(* IEC 61131-3 sources: plc_simulator/services/codesys/POUs/SIM, 13 files *)

(* ---- SIM_FindStation.st ---- *)
(* ============================================================
 *  SIM_FindStation — Find a station by its number

   Company : Galvatek part of the John Cockerill Group
   Author  : Jarmo Piipponen
   Created : 25.03.2026
   ============================================================
   Direct lookup in Stations[] by station number.
   Returns x_mm (DINT); other fields via VAR_OUTPUT.
   ------------------------------------------------------------
   Changes:
   ============================================================ *)

FUNCTION SIM_FindStation : DINT   (* returns x_mm *)
VAR_INPUT
  station_number : INT;
END_VAR
VAR_OUTPUT
  found           : BOOL;
  skind           : INT;
  device_delay_s  : REAL;
  dropping_time_s : REAL;
END_VAR
VAR_EXTERNAL CONSTANT
    MIN_StationIndex : INT;
    MAX_StationIndex : INT;
END_VAR
VAR_EXTERNAL
  Stations : ARRAY[MIN_StationIndex..MAX_StationIndex] OF UDT_StationType;
END_VAR
VAR
  stn_data : UDT_StationType;
END_VAR

  (* Direct lookup by station number — no loop needed *)
  IF (station_number >= MIN_StationIndex) AND (station_number <= MAX_StationIndex) THEN
    stn_data := Stations[station_number];
    IF stn_data.TankId <> 0 THEN
      found := TRUE;
      SIM_FindStation := stn_data.XPosition;
      skind := stn_data.DryWet;
      device_delay_s := INT_TO_REAL(stn_data.DeviceDelay) / 10.0;
      dropping_time_s := INT_TO_REAL(stn_data.DrippingTime) / 10.0;
      RETURN;
    END_IF;
  END_IF;

  found := FALSE;
  SIM_FindStation := 0;
  skind := 0;
  device_delay_s := 0.0;
  dropping_time_s := 0.0;

END_FUNCTION

(* ---- FB_SIM_ClearConfig.st ---- *)
(* ============================================================
   FB_SIM_ClearConfig — Clear all PLC configuration data

   Company : Galvatek part of the John Cockerill Group
   Author  : Jarmo Piipponen
   Created : 25.03.2026
   ============================================================
   Called by PLC_PRG when Gateway sends cmd=3 (clear_all).
   Zeroes out all stations, transporter configs, transporter
   states and units so the PLC is ready for fresh config upload.
   ------------------------------------------------------------
   Changes:
   ============================================================ *)

FUNCTION_BLOCK FB_SIM_ClearConfig
VAR_EXTERNAL CONSTANT
    MAX_TRANSPORTERS    : INT;
    MAX_STATIONS_PER_STEP       : INT;
    MAX_STEPS_PER_PROGRAM       : INT;
    MAX_TASK_QUEUE      : INT;
    MIN_STATION_INDEX : INT;
    MAX_STATION_INDEX   : INT;
    MAX_UNITS           : INT;
    DEP_MAX_WAITING     : INT;
    NOT_PROCESSED       : INT;
END_VAR

VAR_EXTERNAL
  CountStations       : INT;
  Stations         : ARRAY[MIN_STATION_INDEX..MAX_STATION_INDEX] OF UDT_StationType;
  g_station_occupancy     : ARRAY[1..MAX_STATION_INDEX] OF UDT_JC_UnitAtStationType;
  Transporters              : ARRAY[0..MAX_TRANSPORTERS] OF UDT_TransporterType;
  g_transporter      : ARRAY[1..MAX_TRANSPORTERS] OF UDT_TransporterStatusType;
  g_sim_trans        : ARRAY[1..MAX_TRANSPORTERS] OF UDT_JC_SimTransporterType;
  g_dispatched_task  : ARRAY[1..MAX_TRANSPORTERS] OF UDT_JC_DispatchedTaskType;
  g_unit            : ARRAY[1..MAX_UNITS] OF UDT_JC_UnitType;
  g_ntt             : ARRAY[1..MAX_TRANSPORTERS] OF UDT_JC_NttTransporterType;
  g_batch          : ARRAY[1..MAX_UNITS] OF UDT_BatchType;
  TreatmentPrograms         : ARRAY[1..MAX_UNITS] OF UDT_TreatmentProgramType;
  g_avoid_status     : ARRAY[MIN_STATION_INDEX..MAX_STATION_INDEX] OF INT;
  g_schedule         : ARRAY[1..MAX_UNITS] OF UDT_JC_TskScheduleType;
  g_task             : ARRAY[1..MAX_TRANSPORTERS] OF UDT_JC_TskQueueType;
  g_sim_ui_schedule  : ARRAY[1..MAX_UNITS] OF UDT_JC_TskScheduleType;
  g_sim_ui_task      : ARRAY[1..MAX_TRANSPORTERS] OF UDT_JC_TskQueueType;
  g_sim_ui_wait_unit : INT;
  g_sim_ui_wait_reason : INT;
  g_dep_pending      : UDT_JC_DepPendingWriteType;
  g_dep_activated    : BOOL;
  g_tsk_stable       : BOOL;
  g_dep_waiting_count : INT;
  g_dep_waiting       : ARRAY[1..DEP_MAX_WAITING] OF INT;
END_VAR
VAR
  i : INT;
  j : INT;
  k : INT;
END_VAR

(* --- Clear all stations --- *)
FOR i := MIN_STATION_INDEX TO MAX_STATION_INDEX DO
  Stations[i].TankId       := 0;
  Stations[i].IsInUse       := FALSE;
  Stations[i].XPosition    := 0;
  Stations[i].YPosition    := 0;
  Stations[i].ZPosition    := 0;
  Stations[i].DryWet          := 0;
  Stations[i].StationType     := 0;
  Stations[i].DrippingTime := 0;
  Stations[i].DeviceDelay  := 0;
END_FOR;

(* --- Clear all vLocation tracking (transporters 1..MAX_TRANSPORTERS + stations MIN..MAX) --- *)
FOR i := 1 TO MAX_STATION_INDEX DO
  g_station_occupancy[i].UnitId     := 0;
  g_station_occupancy[i].ChangeTime := 0;
END_FOR;
CountStations := 0;

(* --- Clear all transporter configs --- *)
FOR i := 1 TO MAX_TRANSPORTERS DO
  Transporters[i].DrivePosMin   := 0;
  Transporters[i].DrivePosMax   := 0;
  Transporters[i].YMinDriveLimit   := 0;
  Transporters[i].YMaxDriveLimit   := 0;
  Transporters[i].CollisionWidth    := 0;
  Transporters[i].AvoidanceWidth    := 0;
  Transporters[i].Acceleration_X     := 0;
  Transporters[i].Deceleration_X     := 0;
  Transporters[i].SpeedMax_X    := 0;
  Transporters[i].ZPosDown    := 0;
  Transporters[i].ZPosSlowUp := 0;
  Transporters[i].ZPosSlowDown := 0;
  Transporters[i].ZPosSlowEnd := 0;
  Transporters[i].SpeedLiftSlow_Z   := 0;
  Transporters[i].SpeedLiftFast_Z   := 0;
  Transporters[i].DripTrayDelay  := 0;
  FOR j := 1 TO 4 DO
    Transporters[i].TaskArea[j].MinLift := 0;
    Transporters[i].TaskArea[j].MaxLift := 0;
    Transporters[i].TaskArea[j].MinSink := 0;
    Transporters[i].TaskArea[j].MaxSink := 0;
  END_FOR;
END_FOR;

(* --- Clear avoid status --- *)
FOR i := MIN_STATION_INDEX TO MAX_STATION_INDEX DO
  g_avoid_status[i] := 0;
END_FOR;

(* --- Clear all transporter states --- *)
FOR i := 1 TO MAX_TRANSPORTERS DO
  g_transporter[i].IsActive          := FALSE;
  g_transporter[i].Status          := 0;
  g_transporter[i].Phase           := 0;
  g_transporter[i].TaskId         := 0;
  g_transporter[i].LiftStationTarget    := 0;
  g_transporter[i].SinkStationTarget    := 0;
  g_transporter[i].DrippingTime   := 0;
  g_transporter[i].TaskRemainingTime  := 0;
  g_transporter[i].CurrentStation := 0;
  g_transporter[i].XFinalTarget  := 0;
  g_transporter[i].XDriveTarget  := 0;
  g_transporter[i].YFinalTarget  := 0;
  g_transporter[i].YDriveTarget  := 0;
  g_transporter[i].XPosition            := 0;
  g_transporter[i].YPosition            := 0;
  g_transporter[i].ZPosition            := 0;
  g_sim_trans[i].XVelocity           := 0;
  g_sim_trans[i].ZStage         := 0;
  g_sim_trans[i].ZTimer       := 0.0;
  g_transporter[i].IdleStartTime := g_time_s;  (* prevent spurious move-away after clear *)
  g_dispatched_task[i].Active := FALSE;
  g_transporter[i].XMinDriveLimit     := 0;
  g_transporter[i].XMaxDriveLimit     := 0;
END_FOR;

(* --- Clear all units --- *)
FOR i := 1 TO MAX_UNITS DO
  g_unit[i].vLocation := 0;
  g_unit[i].Status   := 0;
  g_unit[i].Target   := 0;
END_FOR;

(* --- Clear NTT destinations --- *)
FOR i := 1 TO MAX_TRANSPORTERS DO
  FOR j := 1 TO 8 DO
    g_ntt[i].Target[j].StationCount := 0;
    g_ntt[i].Target[j].FallbackCount := 0;
    FOR k := 1 TO MAX_STATIONS_PER_STEP DO
      g_ntt[i].Target[j].Stations[k] := 0;
      g_ntt[i].Target[j].FallbackStations[k] := 0;
    END_FOR;
  END_FOR;
END_FOR;

(* --- Clear all batches --- *)
FOR i := 1 TO MAX_UNITS DO
  g_batch[i].BatchCode  := 0;
  g_batch[i].State       := 0;
  g_batch[i].ProgId     := 0;
  g_batch[i].CurStage   := 0;
  g_batch[i].MinTime    := 0;
  g_batch[i].MaxTime    := 0;
  g_batch[i].CalTime    := 0;
  g_batch[i].StartTime  := LINT#0;
END_FOR;

(* --- Clear all treatment programs --- *)
FOR i := 1 TO MAX_UNITS DO
  TreatmentPrograms[i].ProgramId := 0;
  TreatmentPrograms[i].ProgramName := '';
  TreatmentPrograms[i].StepCount := 0;
  FOR j := 0 TO MAX_STEPS_PER_PROGRAM DO
    FOR k := 0 TO 4 DO
      TreatmentPrograms[i].Steps[j].Stations[k] := 0;
    END_FOR;
    TreatmentPrograms[i].Steps[j].StationCount := 0;
    TreatmentPrograms[i].Steps[j].MinTime := 0;
    TreatmentPrograms[i].Steps[j].MaxTime := 0;
    TreatmentPrograms[i].Steps[j].CalTime := 0;
  END_FOR;
END_FOR;

(* --- Clear all schedules (g_schedule) --- *)
FOR i := 1 TO MAX_UNITS DO
  g_schedule[i].StageCount := 0;
  FOR j := 0 TO MAX_STEPS_PER_PROGRAM DO
    g_schedule[i].Stages[j].Station       := 0;
    g_schedule[i].Stages[j].EntryTime    := 0;
    g_schedule[i].Stages[j].ExitTime     := 0;
    g_schedule[i].Stages[j].MinTime      := 0;
    g_schedule[i].Stages[j].CalcTime     := 0;
    g_schedule[i].Stages[j].MaxTime      := 0;
    g_schedule[i].Stages[j].TransferTime := 0;
  END_FOR;
END_FOR;

(* --- Clear all task queues (g_task) --- *)
FOR i := 1 TO MAX_TRANSPORTERS DO
  g_task[i].Count := 0;
  FOR j := 1 TO MAX_TASK_QUEUE DO
    g_task[i].Queue[j].Unit         := 0;
    g_task[i].Queue[j].Stage        := 0;
    g_task[i].Queue[j].LiftStationTarget := 0;
    g_task[i].Queue[j].SinkStationTarget := 0;
    g_task[i].Queue[j].StartTime   := 0;
    g_task[i].Queue[j].FinishTime  := 0;
    g_task[i].Queue[j].CalcTime    := 0;
    g_task[i].Queue[j].MinTime     := 0;
    g_task[i].Queue[j].MaxTime     := 0;
  END_FOR;
END_FOR;

(* --- Clear UI snapshot --- *)
FOR i := 1 TO MAX_UNITS DO
  g_sim_ui_schedule[i].StageCount := 0;
END_FOR;
FOR i := 1 TO MAX_TRANSPORTERS DO
  g_sim_ui_task[i].Count := 0;
END_FOR;
g_sim_ui_wait_unit := 0;
g_sim_ui_wait_reason := 0;

(* --- Clear departure pending write --- *)
g_dep_pending.Valid := FALSE;
g_dep_pending.BatchUnit  := 0;
g_dep_pending.BatchStage := 0;
g_dep_pending.BatchState := NOT_PROCESSED;

(* --- Clear departure scheduler state (previously missing) --- *)
g_dep_activated     := FALSE;
g_tsk_stable        := TRUE;   (* JS: tasksStableFlag starts true on empty line *)
g_dep_waiting_count := 0;
FOR i := 1 TO 5 DO
  g_dep_waiting[i] := 0;
END_FOR;

END_FUNCTION_BLOCK

(* ---- FB_SIM_EventQueue.st ---- *)
(* ============================================================
   FB_SIM_EventQueue — Event message queue handler (OPC UA)

   Company : Galvatek part of the John Cockerill Group
   Author  : Jarmo Piipponen
   Created : 25.03.2026
   ============================================================
   Manages a circular 10-slot event queue (g_event).

   Enqueue: caller writes msg to g_event_pending, sets
   g_event_pending_valid := TRUE. This FB picks it up.

   Dequeue: Gateway reads g_event.Buffer[Head] via OPC UA,
   then writes g_event_ack_seq to acknowledge.

   Called every PLC scan from PLC_PRG.
   ------------------------------------------------------------
   Changes:
   ============================================================ *)

FUNCTION_BLOCK FB_SIM_EventQueue
VAR_EXTERNAL
  g_event               : UDT_JC_EventQueueType;
  g_event_pending       : UDT_JC_EventMsgType;
  g_event_pending_valid : BOOL;
  g_event_ack_seq       : INT;
END_VAR
VAR
  vTail : INT;
END_VAR

(* ── 1. Enqueue: pick up pending message if queue not full ── *)
IF g_event_pending_valid AND g_event.Count < 10 THEN
  vTail := ((g_event.Head - 1 + g_event.Count) MOD 10) + 1;

  g_event_pending.Seq := g_event.NextSeq;
  g_event.NextSeq := g_event.NextSeq + 1;
  IF g_event.NextSeq > 32000 THEN
    g_event.NextSeq := 1;
  END_IF;

  g_event.Buffer[vTail] := g_event_pending;
  g_event.Count := g_event.Count + 1;

  g_event_pending_valid := FALSE;
END_IF;

(* ── 2. Dequeue: check gateway ack for head message ── *)
IF g_event.Count > 0 THEN
  IF g_event_ack_seq = g_event.Buffer[g_event.Head].Seq THEN
    g_event.Head := (g_event.Head MOD 10) + 1;
    g_event.Count := g_event.Count - 1;
  END_IF;
END_IF;

END_FUNCTION_BLOCK

(* ---- FB_SIM_MainCycle.st ---- *)
(* ===========================================================================================
 *  FB_SIM_MainCycle — Simulator main cycle (all SIM-specific logic)
 *
 *  Company : Galvatek part of the John Cockerill Group
 *  Author  : Jarmo Piipponen
 *  Created : 08.04.2026
 *
 * -------------------------------------------------------------------------------------------
 *  Encapsulates everything that is simulation-only and NOT vNeeded in production:
 *    - OPC UA command handler (init / clear)
 *    - System time calculation (g_time_s via offset from gateway sync)
 *    - TWA calculation
 *    - Physics simulation (delta_t + FB_SIM_RunTasks)
 *    - UI schedule snapshot for gateway
 *    - Event queue processing
 *
 *  In production PLC_PRG, this FB is removed entirely.
 *  PLC_PRG only needs: time from real PLC clock, TWA, MainScheduler.
 * ========================================================================================= *)

FUNCTION_BLOCK FB_SIM_MainCycle

(* Introduction of Variables ----------------------------------------------------------------*)

VAR_EXTERNAL CONSTANT
    MAX_TRANSPORTERS        : INT;
    MAX_STATIONS_PER_STEP   : INT;
    MIN_STATION_INDEX        : INT;
    MAX_STATION_INDEX        : INT;
    MAX_UNITS               : INT;
    DEP_MAX_WAITING         : INT;
END_VAR

VAR_EXTERNAL
  CountStations             : INT;
  Stations                  : ARRAY[MIN_STATION_INDEX..MAX_STATION_INDEX] OF UDT_StationType;
  g_station_occupancy       : ARRAY[1..MAX_STATION_INDEX] OF UDT_JC_UnitAtStationType;
  Transporters              : ARRAY[0..MAX_TRANSPORTERS] OF UDT_TransporterType;
  g_transporter             : ARRAY[1..MAX_TRANSPORTERS] OF UDT_TransporterStatusType;
  g_sim_trans               : ARRAY[1..MAX_TRANSPORTERS] OF UDT_JC_SimTransporterType;
  g_unit                    : ARRAY[1..MAX_UNITS] OF UDT_JC_UnitType;
  g_ntt                     : ARRAY[1..MAX_TRANSPORTERS] OF UDT_JC_NttTransporterType;
  g_batch                   : ARRAY[1..MAX_UNITS] OF UDT_BatchType;
  TreatmentPrograms         : ARRAY[1..MAX_UNITS] OF UDT_TreatmentProgramType;
  g_avoid_status            : ARRAY[MIN_STATION_INDEX..MAX_STATION_INDEX] OF INT;
  g_move                    : ARRAY[1..MAX_TRANSPORTERS] OF UDT_JC_MoveTimesType;
  g_schedule                : ARRAY[1..MAX_UNITS] OF UDT_JC_TskScheduleType;
  g_task                    : ARRAY[1..MAX_TRANSPORTERS] OF UDT_JC_TskQueueType;
  g_dep_activated           : BOOL;
  g_tsk_stable              : BOOL;
  g_dep_waiting_count       : INT;
  g_dep_overlap             : UDT_JC_DepOverlapType;
  g_dep_pending             : UDT_JC_DepPendingWriteType;
  g_dep_waiting             : ARRAY[1..DEP_MAX_WAITING] OF INT;
  g_sched_dbg_tsk_phase     : INT;
  g_sched_dbg_dep_phase     : INT;
  g_sim_ui_schedule         : ARRAY[1..MAX_UNITS] OF UDT_JC_TskScheduleType;
  g_sim_ui_task             : ARRAY[1..MAX_TRANSPORTERS] OF UDT_JC_TskQueueType;
  g_sim_ui_wait_unit        : INT;
  g_sim_ui_wait_reason      : INT;
  g_sched_dbg_turn          : INT;
  g_conflict_resolved       : BOOL;
  g_sched_dbg_batch_cnt     : INT;
  g_time_s                  : LINT;
  g_time_100ms              : LINT;
  g_time_offset             : LINT;
  g_time_sync               : LINT;
  g_event                   : UDT_JC_EventQueueType;
  g_event_pending           : UDT_JC_EventMsgType;
  g_event_pending_valid     : BOOL;
  g_event_ack_seq           : INT;
  g_cmd_code                : INT;
  g_cmd_param               : INT;
  g_sched_dbg_dep_cur_wait_unit : INT;
END_VAR

VAR_OUTPUT
  oInitDone               : BOOL;
END_VAR

VAR
  vInitDone                 : BOOL := FALSE;
  i                         : INT;
  vFB_ClearConfig                 : FB_SIM_ClearConfig;
  vFB_RunTasks                 : FB_SIM_RunTasks;
  vFB_EventQueue                 : FB_SIM_EventQueue;
  vNowMs                    : LINT := 0;
  vPrevMs                   : UDINT := 0;
  sim_delta_t               : REAL := 0.02;
  vPrevTskPhase            : INT := 0;
  vPrevDepPhase            : INT := 0;
END_VAR

(* ============================================================
   COMMAND HANDLER — OPC UA (direct, no sequence handshake)
   Gateway writes g_cmd_code + g_cmd_param in one atomic OPC UA
   call. PLC processes when g_cmd_code <> 0 and clears it.
   ============================================================ *)
IF g_cmd_code <> 0 THEN

  IF g_cmd_code = 3 THEN
    (* ── Clear all config data ── *)
    vFB_ClearConfig();
    vInitDone := FALSE;
    CountStations := 0;

  ELSIF g_cmd_code = 2 THEN
    (* ── Finish init: all config vAlready uploaded via OPC UA ── *)
    CountStations := g_cmd_param;

    FOR i := 1 TO MAX_TRANSPORTERS DO
      IF Transporters[i].TaskArea[1].MinLift > 0 THEN
        g_transporter[i].IsActive := TRUE;
        g_transporter[i].Status := 3;  (* auto_idle *)
      ELSE
        g_transporter[i].IsActive := FALSE;
        g_transporter[i].Status := 0;  (* not_used *)
      END_IF;
      g_transporter[i].Phase := 0;
      g_sim_trans[i].ZStage := 0;
      g_sim_trans[i].XVelocity := 0;
      g_sim_trans[i].ZTimer := 0.0;
      g_transporter[i].IdleStartTime := g_time_s;
      g_transporter[i].XMinDriveLimit := Transporters[i].DrivePosMin;
      g_transporter[i].XMaxDriveLimit := Transporters[i].DrivePosMax;

      (* Start position: at own vArea minimum, z=0 *)
      g_transporter[i].XPosition := Transporters[i].DrivePosMin;
      g_transporter[i].ZPosition := 0;
      g_transporter[i].CurrentStation := 0;
    END_FOR;

    vInitDone := TRUE;

    (* Calculate time offset: real unix time - uptime *)
    g_time_offset := g_time_sync - UDINT_TO_LINT(SysTimeGetMs()) / 1000;

    (* Build g_station_occupancy from g_unit[].vLocation so FB_SIM_RunTasks
       can find units on stations via g_station_occupancy[stn].UnitId.
       Gateway writes g_unit[] but not g_station_occupancy[]. *)
    FOR i := 1 TO MAX_UNITS DO
      IF g_unit[i].vLocation >= MIN_STATION_INDEX
         AND g_unit[i].vLocation <= MAX_STATION_INDEX THEN
        g_station_occupancy[g_unit[i].vLocation].UnitId     := i;
        g_station_occupancy[g_unit[i].vLocation].ChangeTime  := g_time_s;
      END_IF;
    END_FOR;

    (* Init event queue *)
    g_event.Head := 1;
    g_event.NextSeq := 1;
    g_event.Count := 0;
  END_IF;

  g_cmd_code := 0;  (* Command processed — clear trigger *)
END_IF;

(* ============================================================
   MAIN TRANSPORT CYCLE — only runs when vInitDone
   ============================================================ *)
IF vInitDone THEN

  (* ── System time: uptime + offset = real unix seconds ── *)
  vNowMs := UDINT_TO_LINT(SysTimeGetMs());
  g_time_s := g_time_offset + vNowMs / 1000;        (* seconds, unix epoch *)
  g_time_100ms := g_time_offset * 10 + vNowMs / 100; (* 0.1s ticks, unix epoch *)

  (* ── Actual cycle time for physics simulation ── *)
  IF vPrevMs > 0 THEN
    sim_delta_t := UDINT_TO_REAL(LINT_TO_UDINT(vNowMs) - vPrevMs) / 1000.0;
  END_IF;
  vPrevMs := LINT_TO_UDINT(vNowMs);

  (* ── Execute transporter tasks (physics simulation) ── *)
  vFB_RunTasks(iRun := vInitDone, iDeltaT := sim_delta_t);

END_IF;  (* vInitDone *)

oInitDone := vInitDone;

(* ── UI schedule snapshot — copy stable data for gateway reads ── *)
IF g_sched_dbg_tsk_phase = 10000 AND vPrevTskPhase <> 10000 THEN
  g_sim_ui_schedule := g_schedule;
  g_sim_ui_task     := g_task;
END_IF;
IF g_sched_dbg_dep_phase = 8000 AND vPrevDepPhase <> 8000 THEN
  g_sim_ui_wait_unit   := 0;
  g_sim_ui_wait_reason := 0;
END_IF;
IF g_sched_dbg_dep_phase = 9000 AND vPrevDepPhase <> 9000 THEN
  g_sim_ui_wait_unit   := g_sched_dbg_dep_cur_wait_unit;
  g_sim_ui_wait_reason := 1;
END_IF;
vPrevTskPhase := g_sched_dbg_tsk_phase;
vPrevDepPhase := g_sched_dbg_dep_phase;

(* ── Event queue — always runs, not gated by vInitDone ── *)
vFB_EventQueue();

END_FUNCTION_BLOCK

(* ---- FB_SIM_RunTasks.st ---- *)
(* ============================================================
   FB_SIM_RunTasks — Simulate transporter task execution

   Company : Galvatek part of the John Cockerill Group
   Author  : Jarmo Piipponen
   Created : 25.03.2026
   ============================================================
   For each active transporter [1..3], checks whether a new task
   has been assigned (task_id <> running_task_id) and executes
   the full transport cycle:

     Phase 0  idle        — waiting for new task
     Phase 1  to_lift     — X-drive towards lift station
     Phase 2  lifting     — Z-lift sequence (stages 1-5)
     Phase 3  to_sink     — X-drive towards sink station
     Phase 4  sinking     — Z-sink sequence (stages 6-8)

   Also maintains current_station (nearest station) every cycle.
   Called once per PLC scan from PLC_PRG.
   ------------------------------------------------------------
   Changes:
   ============================================================ *)

FUNCTION_BLOCK FB_SIM_RunTasks
VAR_INPUT
  iRun     : BOOL;   (* enable — typically vInitDone *)
  iDeltaT : REAL;   (* actual cycle time in seconds *)
END_VAR
VAR_EXTERNAL CONSTANT
    MAX_TRANSPORTERS    : INT;
    MAX_UNITS           : INT;
    MAX_STEPS_PER_PROGRAM          : INT;
    MIN_STATION_INDEX : INT;
    MAX_STATION_INDEX   : INT;
    IN_PROCESS          : INT;
END_VAR

VAR_EXTERNAL
  g_transporter  : ARRAY[1..MAX_TRANSPORTERS] OF UDT_TransporterStatusType;
  g_sim_trans    : ARRAY[1..MAX_TRANSPORTERS] OF UDT_JC_SimTransporterType;
  Stations      : ARRAY[MIN_STATION_INDEX..MAX_STATION_INDEX] OF UDT_StationType;
  g_station_occupancy  : ARRAY[1..MAX_STATION_INDEX] OF UDT_JC_UnitAtStationType;
  Transporters          : ARRAY[0..MAX_TRANSPORTERS] OF UDT_TransporterType;
  g_move         : ARRAY[1..MAX_TRANSPORTERS] OF UDT_JC_MoveTimesType;
  g_actual_move  : ARRAY[1..MAX_TRANSPORTERS] OF UDT_JC_ActualMoveTimeType;
  g_unit         : ARRAY[1..MAX_UNITS] OF UDT_JC_UnitType;
  g_batch        : ARRAY[1..MAX_UNITS] OF UDT_BatchType;
  TreatmentPrograms      : ARRAY[1..MAX_UNITS] OF UDT_TreatmentProgramType;
  g_time_s       : LINT;
  g_event_pending       : UDT_JC_EventMsgType;
  g_event_pending_valid : BOOL;
  g_dispatched_task     : ARRAY[1..MAX_TRANSPORTERS] OF UDT_JC_DispatchedTaskType;
END_VAR
VAR
  i            : INT;
  vIdx          : INT;
  (* Physics FB instances — one per transporter (MATIEC needs separate instances) *)
  fb_x1        : FB_SIM_XMotion;
  fb_x2        : FB_SIM_XMotion;
  fb_x3        : FB_SIM_XMotion;
  fb_z1        : FB_SIM_ZMotion;
  fb_z2        : FB_SIM_ZMotion;
  fb_z3        : FB_SIM_ZMotion;
  (* Temp vars for VAR_IN_OUT passing *)
  vTmpX        : DINT;
  vTmpVx       : DINT;
  vTmpZ        : DINT;
  vTmpZs       : INT;
  vTmpZt       : REAL;
  arrived_x    : BOOL;
  at_station   : BOOL;    (* TRUE only when actually at station, not just at drive limit *)
  arrived_z    : BOOL;
  vStationKind : INT;
  device_delay : REAL;
  vDropTime    : REAL;
  vPickUnitId : INT;     (* unit_id picked up from lift station *)
  vXferTotal   : REAL;    (* transfer time for UI progress bar *)
  vSinkUnitId : INT;     (* unit_id being placed at sink station *)
  (* Nearest-station calculation *)
  vNearestNum  : INT;
  vMinDist     : DINT;
  dx           : DINT;
  (* Actual move time tracker — now FC FC_STC_TrackMoveTimes, no instance vNeeded *)
  (* Unit vLocation update — now FC FC_STC_UpdateUnitLocation, no instance vNeeded *)
  (* Event helpers *)
  evt_unit     : INT;
  evt_diff     : LINT;
  (* Treatment time wait *)
  vCanLift       : BOOL;
  vLiftUid       : INT;      (* unit at lift station *)
  treat_cal      : DINT;      (* treatment cal_time for current stage *)
  treat_elapsed  : LINT;     (* seconds spent at lift station *)
  (* ── TASK_COMPLETE event: vPhase timestamps per transporter ── *)
  ts_task_start  : ARRAY[1..3] OF LINT;  (* Phase 0→1: task accepted *)
  ts_at_lift     : ARRAY[1..3] OF LINT;  (* Phase 1 at_station: arrived at lift *)
  ts_lift_begin  : ARRAY[1..3] OF LINT;  (* Phase 1→2: vCanLift, begin lift *)
  ts_lift_done   : ARRAY[1..3] OF LINT;  (* Phase 2→3: lift complete *)
  ts_at_sink     : ARRAY[1..3] OF LINT;  (* Phase 3→4: arrived at sink *)
  (* TASK_COMPLETE temp vars *)
  dd_lift_s      : INT;   (* lift device_delay in seconds *)
  dropping_s     : INT;   (* dropping/valutus time in seconds *)
  trip_s         : INT;   (* drip tray vDelay in seconds, 0 if not used *)
  vDurNosto      : INT;   (* computed nosto vDuration *)
  vDurLasku      : INT;   (* computed lasku vDuration *)
END_VAR

IF NOT iRun THEN
  RETURN;
END_IF;

FOR i := 1 TO MAX_TRANSPORTERS DO
  IF g_transporter[i].IsActive THEN

  (* ── Phase 0 → 1: Accept new task ───────────────────────── *)
  IF (g_transporter[i].Phase = 0)
     AND g_dispatched_task[i].Active THEN
    g_transporter[i].XFinalTarget := g_dispatched_task[i].LiftX;
    g_transporter[i].Status := 4;  (* auto_run — must be set before TrackMoveTimes *)
    g_transporter[i].Phase := 1;
    FC_STC_TrackMoveTimes(iTrans := i, iPrev := 0, iNew := 1);
    g_sim_trans[i].ZStage := 0;
    g_sim_trans[i].ZTimer := 0.0;
    (* Record task start timestamp *)
    ts_task_start[i] := g_time_s;
    ts_at_lift[i]    := LINT#0;

  (* ── Phase 1: Drive X towards lift station ──────────────── *)
  ELSIF g_transporter[i].Phase = 1 THEN
    vTmpX  := g_transporter[i].XPosition;
    vTmpVx := g_sim_trans[i].XVelocity;
    IF i = 1 THEN
      fb_x1(
        delta_t  := iDeltaT,
        x_target := g_transporter[i].XFinalTarget,
        x_min    := g_transporter[i].XMinDriveLimit,
        x_max    := g_transporter[i].XMaxDriveLimit,
        v_max    := Transporters[i].SpeedMax_X,
        t_acc    := Transporters[i].Acceleration_X,
        t_dec    := Transporters[i].Deceleration_X,
        x_pos    := vTmpX,
        v_x      := vTmpVx
      );
      arrived_x := fb_x1.arrived;
      g_transporter[i].XDriveTarget := fb_x1.x_drive;
    ELSIF i = 2 THEN
      fb_x2(
        delta_t  := iDeltaT,
        x_target := g_transporter[i].XFinalTarget,
        x_min    := g_transporter[i].XMinDriveLimit,
        x_max    := g_transporter[i].XMaxDriveLimit,
        v_max    := Transporters[i].SpeedMax_X,
        t_acc    := Transporters[i].Acceleration_X,
        t_dec    := Transporters[i].Deceleration_X,
        x_pos    := vTmpX,
        v_x      := vTmpVx
      );
      arrived_x := fb_x2.arrived;
      g_transporter[i].XDriveTarget := fb_x2.x_drive;
    ELSIF i = 3 THEN
      fb_x3(
        delta_t  := iDeltaT,
        x_target := g_transporter[i].XFinalTarget,
        x_min    := g_transporter[i].XMinDriveLimit,
        x_max    := g_transporter[i].XMaxDriveLimit,
        v_max    := Transporters[i].SpeedMax_X,
        t_acc    := Transporters[i].Acceleration_X,
        t_dec    := Transporters[i].Deceleration_X,
        x_pos    := vTmpX,
        v_x      := vTmpVx
      );
      arrived_x := fb_x3.arrived;
      g_transporter[i].XDriveTarget := fb_x3.x_drive;
    END_IF;
    g_transporter[i].XPosition  := vTmpX;
    g_sim_trans[i].XVelocity := vTmpVx;

    (* Only transition when actually at station, not just at drive limit *)
    at_station := arrived_x
                  AND (ABS(g_transporter[i].XPosition - g_transporter[i].XFinalTarget) <= 6);
    IF at_station THEN
      g_transporter[i].CurrentStation := g_transporter[i].LiftStationTarget;

      (* ── Move-away arrival: Status=3 means idle repositioning, not a real task ── *)
      IF g_transporter[i].Status = 3 THEN
        g_transporter[i].Phase := 0;
        g_transporter[i].IdleStartTime := g_time_s;
        FC_STC_TrackMoveTimes(iTrans := i, iPrev := 1, iNew := 0);
      ELSE
      (* Record arrival at lift station (first time only) *)
      IF ts_at_lift[i] = LINT#0 THEN
        ts_at_lift[i] := g_time_s;
      END_IF;

      (* ── Wait for treatment time AND device_delay before lifting ──
         Z-movement starts when the LONGER of two has elapsed:
         1. Remaining treatment time (unit must finish treatment)
         2. Station device_delay (vCovers must be open)
         Both timers run simultaneously from transporter arrival.
         This matches JS behavior: max(treatment, device_delay). *)
      vCanLift := TRUE;
      device_delay := INT_TO_REAL(g_dispatched_task[i].LiftDeviceDelay_x10) / 10.0;
      vDropTime := INT_TO_REAL(g_dispatched_task[i].DroppingTime_x10) / 10.0;

      (* Check treatment time *)
      vLiftUid := g_station_occupancy[g_transporter[i].LiftStationTarget].UnitId;
      IF vLiftUid >= 1 AND vLiftUid <= MAX_UNITS THEN
        IF g_batch[vLiftUid].State = IN_PROCESS
           AND g_batch[vLiftUid].CurStage >= 1
           AND g_batch[vLiftUid].CurStage <= MAX_STEPS_PER_PROGRAM THEN
          treat_cal := TreatmentPrograms[vLiftUid].Steps[g_batch[vLiftUid].CurStage].CalTime;
          IF treat_cal > 0 THEN
            treat_elapsed := g_time_s - g_station_occupancy[g_transporter[i].LiftStationTarget].ChangeTime;
            IF treat_elapsed < DINT_TO_LINT(treat_cal) THEN
              vCanLift := FALSE;
            END_IF;
          END_IF;
        END_IF;
      END_IF;

      (* Check device_delay — vCovers must have had time to open since arrival *)
      IF vCanLift AND device_delay > 0.0 THEN
        IF LINT_TO_REAL(g_time_s - ts_at_lift[i]) < device_delay THEN
          vCanLift := FALSE;
        END_IF;
      END_IF;

      IF vCanLift THEN
      (* Record lift begin timestamp *)
      ts_lift_begin[i] := g_time_s;
      (* vDropTime vAlready captured by STC_FindStation above *)
      (* Skip stage 1 — device_delay vAlready overlapped above.
         Z-movement starts immediately (stage 2).
         dropping_time and drip_tray_delay happen at the TOP. *)
      g_transporter[i].ZPosition := 0;
      g_sim_trans[i].ZTimer := 0.0;
      g_sim_trans[i].ZStage := 2;
      g_transporter[i].Phase := 2;
      FC_STC_TrackMoveTimes(iTrans := i, iPrev := 1, iNew := 2);

      (* ── Calculate transfer time (used by event + batch times) ── *)
      vXferTotal := DINT_TO_REAL(g_dispatched_task[i].TransferTime_x10) / 10.0;
      IF vXferTotal < 5.0 THEN vXferTotal := 60.0; END_IF;

      (* ── Emit LIFT event (msg_type=2) ── *)
      evt_unit := g_station_occupancy[g_transporter[i].LiftStationTarget].UnitId;
      IF NOT g_event_pending_valid AND evt_unit >= 1 THEN
        g_event_pending.MsgType := 2;
        g_event_pending.TsHi := LINT_TO_UINT(g_time_s / LINT#65536);
        g_event_pending.TsLo := LINT_TO_UINT(g_time_s MOD LINT#65536);
        g_event_pending.Payload[1]  := LINT_TO_INT(g_transporter[i].TaskId / LINT#65536);   (* TaskId_Hi *)
        g_event_pending.Payload[2]  := LINT_TO_INT(g_transporter[i].TaskId MOD LINT#65536);  (* TaskId_Lo *)
        g_event_pending.Payload[3]  := i;
        g_event_pending.Payload[4]  := evt_unit;
        g_event_pending.Payload[5]  := g_transporter[i].LiftStationTarget;
        g_event_pending.Payload[6]  := g_batch[evt_unit].BatchCode;
        g_event_pending.Payload[7]  := g_batch[evt_unit].CurStage;
        evt_diff := g_time_s - g_station_occupancy[g_transporter[i].LiftStationTarget].ChangeTime;
        IF evt_diff > LINT#32000 THEN
          g_event_pending.Payload[8] := 32000;
        ELSE
          g_event_pending.Payload[8] := LINT_TO_INT(evt_diff);
        END_IF;
        (* ── Original program calc/min/max for this stage ── *)
        (* g_sim_trans holds dispatch-time scheduler values which may differ
           from the treatment program originals. Read directly from TreatmentPrograms
           using the batch's current stage (CurStage=1-based program index). *)
        IF g_batch[evt_unit].CurStage >= 1 AND g_batch[evt_unit].CurStage <= 30 THEN
          g_event_pending.Payload[9]  := DINT_TO_INT(TreatmentPrograms[evt_unit].Steps[g_batch[evt_unit].CurStage].CalTime);
          g_event_pending.Payload[10] := DINT_TO_INT(TreatmentPrograms[evt_unit].Steps[g_batch[evt_unit].CurStage].MinTime);
          g_event_pending.Payload[11] := DINT_TO_INT(TreatmentPrograms[evt_unit].Steps[g_batch[evt_unit].CurStage].MaxTime);
        ELSE
          (* Stage 0 (pickup) — no program step *)
          g_event_pending.Payload[9]  := 0;
          g_event_pending.Payload[10] := 0;
          g_event_pending.Payload[11] := 0;
        END_IF;
        g_event_pending.Payload[12] := REAL_TO_INT(vXferTotal);
        g_event_pending_valid := TRUE;
      END_IF;

      (* Unit moves from lift station → transporter *)
      vPickUnitId := g_station_occupancy[g_transporter[i].LiftStationTarget].UnitId;
      IF vPickUnitId >= 1 THEN
        FC_STC_UpdateUnitLocation(iUnit := vPickUnitId, iLocation := i, iNttPrimary := 0);

        (* Set batch transfer times for UI progress bar — matches JS behavior *)
        g_batch[vPickUnitId].StartTime := g_time_s;
        g_batch[vPickUnitId].CalTime   := REAL_TO_DINT(vXferTotal);
        g_batch[vPickUnitId].MinTime   := g_batch[vPickUnitId].CalTime;
        g_batch[vPickUnitId].MaxTime   := 600;
      END_IF;
      END_IF;  (* vCanLift *)
      END_IF;  (* Status=3 ELSE branch *)
    END_IF;
    (* If arrived_x but not at_station → at drive limit, wait for clearance *)

  (* ── Phase 2: Lift Z at lift station ────────────────────── *)
  ELSIF g_transporter[i].Phase = 2 THEN
    vStationKind := g_dispatched_task[i].LiftKind;
    vTmpZ  := g_transporter[i].ZPosition;
    vTmpZs := g_sim_trans[i].ZStage;
    vTmpZt := g_sim_trans[i].ZTimer;
    IF i = 1 THEN
      fb_z1(
        delta_t       := iDeltaT,
        vStationKind  := vStationKind,
        ZPosDown        := Transporters[i].ZPosDown,
        ZPosUp          := 0,
        ZPosSlowUp      := Transporters[i].ZPosSlowUp,
        ZPosSlowDown    := Transporters[i].ZPosSlowDown,
        ZPosSlowEnd     := Transporters[i].ZPosSlowEnd,
        SpeedLiftSlow_Z := Transporters[i].SpeedLiftSlow_Z,
        SpeedLiftFast_Z := Transporters[i].SpeedLiftFast_Z,
        DripTrayDelay   := Transporters[i].DripTrayDelay,
        DroppingTime    := g_dispatched_task[i].DroppingTime_x10,
        z_mm          := vTmpZ,
        z_stage       := vTmpZs,
        z_timer_s     := vTmpZt
      );
      arrived_z := fb_z1.vDone;
    ELSIF i = 2 THEN
      fb_z2(
        delta_t       := iDeltaT,
        vStationKind  := vStationKind,
        ZPosDown        := Transporters[i].ZPosDown,
        ZPosUp          := 0,
        ZPosSlowUp      := Transporters[i].ZPosSlowUp,
        ZPosSlowDown    := Transporters[i].ZPosSlowDown,
        ZPosSlowEnd     := Transporters[i].ZPosSlowEnd,
        SpeedLiftSlow_Z := Transporters[i].SpeedLiftSlow_Z,
        SpeedLiftFast_Z := Transporters[i].SpeedLiftFast_Z,
        DripTrayDelay   := Transporters[i].DripTrayDelay,
        DroppingTime    := g_dispatched_task[i].DroppingTime_x10,
        z_mm          := vTmpZ,
        z_stage       := vTmpZs,
        z_timer_s     := vTmpZt
      );
      arrived_z := fb_z2.vDone;
    ELSIF i = 3 THEN
      fb_z3(
        delta_t       := iDeltaT,
        vStationKind  := vStationKind,
        ZPosDown        := Transporters[i].ZPosDown,
        ZPosUp          := 0,
        ZPosSlowUp      := Transporters[i].ZPosSlowUp,
        ZPosSlowDown    := Transporters[i].ZPosSlowDown,
        ZPosSlowEnd     := Transporters[i].ZPosSlowEnd,
        SpeedLiftSlow_Z := Transporters[i].SpeedLiftSlow_Z,
        SpeedLiftFast_Z := Transporters[i].SpeedLiftFast_Z,
        DripTrayDelay   := Transporters[i].DripTrayDelay,
        DroppingTime    := g_dispatched_task[i].DroppingTime_x10,
        z_mm          := vTmpZ,
        z_stage       := vTmpZs,
        z_timer_s     := vTmpZt
      );
      arrived_z := fb_z3.vDone;
    END_IF;
    g_transporter[i].ZPosition      := vTmpZ;
    g_sim_trans[i].ZStage   := vTmpZs;
    g_sim_trans[i].ZTimer := vTmpZt;
    IF arrived_z THEN
      (* Record lift vDone timestamp *)
      ts_lift_done[i] := g_time_s;
      g_transporter[i].XFinalTarget := g_dispatched_task[i].SinkX;
      g_transporter[i].Phase := 3;
      FC_STC_TrackMoveTimes(iTrans := i, iPrev := 2, iNew := 3);
    END_IF;

  (* ── Phase 3: Drive X towards sink station ─────────────── *)
  ELSIF g_transporter[i].Phase = 3 THEN
    vTmpX  := g_transporter[i].XPosition;
    vTmpVx := g_sim_trans[i].XVelocity;
    IF i = 1 THEN
      fb_x1(
        delta_t  := iDeltaT,
        x_target := g_transporter[i].XFinalTarget,
        x_min    := g_transporter[i].XMinDriveLimit,
        x_max    := g_transporter[i].XMaxDriveLimit,
        v_max    := Transporters[i].SpeedMax_X,
        t_acc    := Transporters[i].Acceleration_X,
        t_dec    := Transporters[i].Deceleration_X,
        x_pos    := vTmpX,
        v_x      := vTmpVx
      );
      arrived_x := fb_x1.arrived;
      g_transporter[i].XDriveTarget := fb_x1.x_drive;
    ELSIF i = 2 THEN
      fb_x2(
        delta_t  := iDeltaT,
        x_target := g_transporter[i].XFinalTarget,
        x_min    := g_transporter[i].XMinDriveLimit,
        x_max    := g_transporter[i].XMaxDriveLimit,
        v_max    := Transporters[i].SpeedMax_X,
        t_acc    := Transporters[i].Acceleration_X,
        t_dec    := Transporters[i].Deceleration_X,
        x_pos    := vTmpX,
        v_x      := vTmpVx
      );
      arrived_x := fb_x2.arrived;
      g_transporter[i].XDriveTarget := fb_x2.x_drive;
    ELSIF i = 3 THEN
      fb_x3(
        delta_t  := iDeltaT,
        x_target := g_transporter[i].XFinalTarget,
        x_min    := g_transporter[i].XMinDriveLimit,
        x_max    := g_transporter[i].XMaxDriveLimit,
        v_max    := Transporters[i].SpeedMax_X,
        t_acc    := Transporters[i].Acceleration_X,
        t_dec    := Transporters[i].Deceleration_X,
        x_pos    := vTmpX,
        v_x      := vTmpVx
      );
      arrived_x := fb_x3.arrived;
      g_transporter[i].XDriveTarget := fb_x3.x_drive;
    END_IF;
    g_transporter[i].XPosition  := vTmpX;
    g_sim_trans[i].XVelocity := vTmpVx;

    (* Only transition when actually at station, not just at drive limit *)
    at_station := arrived_x
                  AND (ABS(g_transporter[i].XPosition - g_transporter[i].XFinalTarget) <= 6);
    IF at_station THEN
      g_transporter[i].CurrentStation := g_transporter[i].SinkStationTarget;
      (* Record arrival at sink timestamp *)
      ts_at_sink[i] := g_time_s;
      device_delay := INT_TO_REAL(g_dispatched_task[i].SinkDeviceDelay_x10) / 10.0;
      g_sim_trans[i].ZTimer := device_delay + INT_TO_REAL(g_dispatched_task[i].DripTrayDelay_x10) / 10.0;
      g_sim_trans[i].ZStage := 6;
      g_transporter[i].Phase := 4;
      FC_STC_TrackMoveTimes(iTrans := i, iPrev := 3, iNew := 4);
    END_IF;
    (* If arrived_x but not at_station → at drive limit, wait for clearance *)

  (* ── Phase 4: Sink Z at sink station ───────────────────── *)
  ELSIF g_transporter[i].Phase = 4 THEN
    vStationKind := g_dispatched_task[i].SinkKind;
    vTmpZ  := g_transporter[i].ZPosition;
    vTmpZs := g_sim_trans[i].ZStage;
    vTmpZt := g_sim_trans[i].ZTimer;
    IF i = 1 THEN
      fb_z1(
        delta_t       := iDeltaT,
        vStationKind  := vStationKind,
        ZPosDown        := Transporters[i].ZPosDown,
        ZPosUp          := 0,
        ZPosSlowUp      := Transporters[i].ZPosSlowUp,
        ZPosSlowDown    := Transporters[i].ZPosSlowDown,
        ZPosSlowEnd     := Transporters[i].ZPosSlowEnd,
        SpeedLiftSlow_Z := Transporters[i].SpeedLiftSlow_Z,
        SpeedLiftFast_Z := Transporters[i].SpeedLiftFast_Z,
        DripTrayDelay   := Transporters[i].DripTrayDelay,
        DroppingTime    := 0,
        z_mm          := vTmpZ,
        z_stage       := vTmpZs,
        z_timer_s     := vTmpZt
      );
      arrived_z := fb_z1.vDone;
    ELSIF i = 2 THEN
      fb_z2(
        delta_t       := iDeltaT,
        vStationKind  := vStationKind,
        ZPosDown        := Transporters[i].ZPosDown,
        ZPosUp          := 0,
        ZPosSlowUp      := Transporters[i].ZPosSlowUp,
        ZPosSlowDown    := Transporters[i].ZPosSlowDown,
        ZPosSlowEnd     := Transporters[i].ZPosSlowEnd,
        SpeedLiftSlow_Z := Transporters[i].SpeedLiftSlow_Z,
        SpeedLiftFast_Z := Transporters[i].SpeedLiftFast_Z,
        DripTrayDelay   := Transporters[i].DripTrayDelay,
        DroppingTime    := 0,
        z_mm          := vTmpZ,
        z_stage       := vTmpZs,
        z_timer_s     := vTmpZt
      );
      arrived_z := fb_z2.vDone;
    ELSIF i = 3 THEN
      fb_z3(
        delta_t       := iDeltaT,
        vStationKind  := vStationKind,
        ZPosDown        := Transporters[i].ZPosDown,
        ZPosUp          := 0,
        ZPosSlowUp      := Transporters[i].ZPosSlowUp,
        ZPosSlowDown    := Transporters[i].ZPosSlowDown,
        ZPosSlowEnd     := Transporters[i].ZPosSlowEnd,
        SpeedLiftSlow_Z := Transporters[i].SpeedLiftSlow_Z,
        SpeedLiftFast_Z := Transporters[i].SpeedLiftFast_Z,
        DripTrayDelay   := Transporters[i].DripTrayDelay,
        DroppingTime    := 0,
        z_mm          := vTmpZ,
        z_stage       := vTmpZs,
        z_timer_s     := vTmpZt
      );
      arrived_z := fb_z3.vDone;
    END_IF;
    g_transporter[i].ZPosition      := vTmpZ;
    g_sim_trans[i].ZStage   := vTmpZs;
    g_sim_trans[i].ZTimer := vTmpZt;
    IF arrived_z THEN
      (* ── Emit TASK_COMPLETE event (msg_type=3) before Phase reset ── *)
      IF NOT g_event_pending_valid THEN
        (* Config-based sub-vPhase durations *)
        dropping_s := g_transporter[i].DrippingTime / 10;
        IF Transporters[i].DripTrayInUse THEN
          trip_s := Transporters[i].DripTrayDelay / 10;
        ELSE
          trip_s := 0;
        END_IF;
        (* Nosto = total lift vPhase - dropping - trip_close
           device_delay no longer in lift vPhase (overlapped in Phase 1) *)
        vDurNosto := LINT_TO_INT(ts_lift_done[i] - ts_lift_begin[i])
                     - dropping_s - trip_s;
        IF vDurNosto < 0 THEN vDurNosto := 0; END_IF;
        (* Lasku = total sink vPhase - device_delay - trip_open *)
        dd_lift_s := g_dispatched_task[i].SinkDeviceDelay_x10 / 10;
        vDurLasku := LINT_TO_INT(g_time_s - ts_at_sink[i]) - dd_lift_s - trip_s;
        IF vDurLasku < 0 THEN vDurLasku := 0; END_IF;

        g_event_pending.MsgType := 3;
        g_event_pending.TsHi := LINT_TO_UINT(g_time_s / LINT#65536);
        g_event_pending.TsLo := LINT_TO_UINT(g_time_s MOD LINT#65536);
        g_event_pending.Payload[1]  := LINT_TO_INT(g_transporter[i].TaskId / LINT#65536);   (* TaskId_Hi *)
        g_event_pending.Payload[2]  := LINT_TO_INT(g_transporter[i].TaskId MOD LINT#65536);  (* TaskId_Lo *)
        g_event_pending.Payload[3]  := i;                                                     (* transporter *)
        g_event_pending.Payload[4]  := LINT_TO_INT(ts_at_lift[i] - ts_task_start[i]);         (* siirto nostoasemalle *)
        g_event_pending.Payload[5]  := LINT_TO_INT(ts_lift_begin[i] - ts_at_lift[i]);         (* odotus ennen nostoa (max(treat,dev_delay)) *)
        g_event_pending.Payload[6]  := vDurNosto;                                             (* nosto *)
        g_event_pending.Payload[7]  := dropping_s;                                            (* valutus *)
        g_event_pending.Payload[8]  := trip_s;                                                (* trip close *)
        g_event_pending.Payload[9]  := LINT_TO_INT(ts_at_sink[i] - ts_lift_done[i]);          (* siirto laskuasemalle *)
        g_event_pending.Payload[10] := trip_s;                                                (* trip open *)
        g_event_pending.Payload[11] := vDurLasku;                                             (* lasku *)
        g_event_pending.Payload[12] := LINT_TO_INT(g_time_s - ts_task_start[i]);              (* total *)
        g_event_pending_valid := TRUE;
      END_IF;

      (* Unit moves from transporter → sink station *)
      vSinkUnitId := g_station_occupancy[i].UnitId;
      IF vSinkUnitId >= 1 THEN
        FC_STC_UpdateUnitLocation(iUnit := vSinkUnitId, iLocation := g_transporter[i].SinkStationTarget, iNttPrimary := g_dispatched_task[i].NttPrimary);
      END_IF;

      g_transporter[i].Phase := 0;
      g_transporter[i].CurrentTaskFinishTime := 0;
      g_dispatched_task[i].Active := FALSE;
      FC_STC_TrackMoveTimes(iTrans := i, iPrev := 4, iNew := 0);
      g_transporter[i].Status := 3;  (* auto_idle *)
      g_transporter[i].IdleStartTime := g_time_s;  (* move-away idle timer *)

    END_IF;
  END_IF;  (* ELSIF chain: phases 0→1→2→3→4 *)

  (* ── Phase 0 idle: drive back inside limits if outside ────── *)
  IF g_transporter[i].Phase = 0 THEN
    vTmpX  := g_transporter[i].XPosition;
    vTmpVx := g_sim_trans[i].XVelocity;
    (* Use current position as target — XMotion will clamp to nearest limit if outside *)
    IF i = 1 THEN
      fb_x1(
        delta_t  := iDeltaT,
        x_target := vTmpX,
        x_min    := g_transporter[i].XMinDriveLimit,
        x_max    := g_transporter[i].XMaxDriveLimit,
        v_max    := Transporters[i].SpeedMax_X,
        t_acc    := Transporters[i].Acceleration_X,
        t_dec    := Transporters[i].Deceleration_X,
        x_pos    := vTmpX,
        v_x      := vTmpVx
      );
    ELSIF i = 2 THEN
      fb_x2(
        delta_t  := iDeltaT,
        x_target := vTmpX,
        x_min    := g_transporter[i].XMinDriveLimit,
        x_max    := g_transporter[i].XMaxDriveLimit,
        v_max    := Transporters[i].SpeedMax_X,
        t_acc    := Transporters[i].Acceleration_X,
        t_dec    := Transporters[i].Deceleration_X,
        x_pos    := vTmpX,
        v_x      := vTmpVx
      );
    ELSIF i = 3 THEN
      fb_x3(
        delta_t  := iDeltaT,
        x_target := vTmpX,
        x_min    := g_transporter[i].XMinDriveLimit,
        x_max    := g_transporter[i].XMaxDriveLimit,
        v_max    := Transporters[i].SpeedMax_X,
        t_acc    := Transporters[i].Acceleration_X,
        t_dec    := Transporters[i].Deceleration_X,
        x_pos    := vTmpX,
        v_x      := vTmpVx
      );
    END_IF;
    g_transporter[i].XPosition  := vTmpX;
    g_sim_trans[i].XVelocity := vTmpVx;
  END_IF;

  (* ── Nearest station tracking ──────────────────────────── *)
  vMinDist := 999999999;
  vNearestNum := g_transporter[i].CurrentStation;
  FOR vIdx := MIN_STATION_INDEX TO MAX_STATION_INDEX DO
    IF Stations[vIdx].TankId <> 0 THEN
      dx := Stations[vIdx].XPosition - g_transporter[i].XPosition;
      IF ABS(dx) < vMinDist THEN
        vMinDist := ABS(dx);
        vNearestNum := vIdx;
      END_IF;
    END_IF;
  END_FOR;
  g_transporter[i].CurrentStation := vNearestNum;

  END_IF;  (* active *)
END_FOR;

END_FUNCTION_BLOCK

(* ---- FB_SIM_XMotion.st ---- *)
(* ============================================================
   FB_SIM_XMotion — Horizontal motion with accel / decel

   Company : Galvatek part of the John Cockerill Group
   Author  : Jarmo Piipponen
   Created : 25.03.2026
   ============================================================
   Trapezoidal velocity profile: accelerate, cruise, decelerate.
   Clamps position to [x_min..x_max] drive limits.
   VAR_IN_OUT: x_pos, v_x (modified in place).
   ------------------------------------------------------------
   Changes:
   ============================================================ *)

FUNCTION_BLOCK FB_SIM_XMotion
VAR_INPUT
  delta_t  : REAL;     (* cycle time s — simulation internal *)
  x_target : DINT;     (* target X mm *)
  x_min    : DINT;     (* TWA lower limit mm *)
  x_max    : DINT;     (* TWA upper limit mm *)
  v_max    : DINT;     (* max velocity mm/s *)
  t_acc    : DINT;     (* acceleration time ×10 = tenths of second *)
  t_dec    : DINT;     (* deceleration time ×10 = tenths of second *)
END_VAR
VAR_IN_OUT
  x_pos : DINT;        (* current X position mm *)
  v_x   : DINT;        (* current X velocity mm/s *)
END_VAR
VAR_OUTPUT
  arrived : BOOL;
  x_drive : DINT;      (* actual drive target after limit clamping *)
END_VAR
VAR
  (* Internal REAL copies for physics integration *)
  r_target     : REAL;
  r_min        : REAL;
  r_max        : REAL;
  r_vmax       : REAL;
  r_tacc       : REAL;
  r_tdec       : REAL;
  r_pos        : REAL;
  r_vel        : REAL;
  drive_target : REAL;
  vDistance     : REAL;
  dir          : REAL;
  a_acc        : REAL;
  a_dec        : REAL;
  brake_dist   : REAL;
  vNewVel      : REAL;
  vTravel       : REAL;
END_VAR
  (* Convert DINT/INT inputs to REAL for physics *)
  r_target := DINT_TO_REAL(x_target);
  r_min    := DINT_TO_REAL(x_min);
  r_max    := DINT_TO_REAL(x_max);
  r_vmax   := DINT_TO_REAL(v_max);
  r_tacc   := DINT_TO_REAL(t_acc) / 10.0;
  r_tdec   := DINT_TO_REAL(t_dec) / 10.0;
  r_pos    := DINT_TO_REAL(x_pos);
  r_vel    := DINT_TO_REAL(v_x);

  IF (r_max > r_min) THEN
    IF r_pos < r_min THEN
      drive_target := r_min;
    ELSIF r_pos > r_max THEN
      drive_target := r_max;
    ELSE
      IF r_target < r_min THEN
        drive_target := r_min;
      ELSIF r_target > r_max THEN
        drive_target := r_max;
      ELSE
        drive_target := r_target;
      END_IF;
    END_IF;
  ELSE
    drive_target := r_target;
  END_IF;

  x_drive := REAL_TO_DINT(drive_target);

  arrived := ABS(r_pos - drive_target) <= 3.0;
  IF arrived THEN
    x_pos := REAL_TO_DINT(drive_target);
    v_x := 0;
    RETURN;
  END_IF;

  IF r_tacc <= 0.0 THEN r_tacc := 0.001; END_IF;
  IF r_tdec <= 0.0 THEN r_tdec := 0.001; END_IF;
  IF r_vmax < 0.0 THEN r_vmax := 0.0; END_IF;

  a_acc := r_vmax / r_tacc;
  a_dec := r_vmax / r_tdec;

  dir := 1.0;
  IF drive_target < r_pos THEN
    dir := -1.0;
  END_IF;

  vDistance := ABS(drive_target - r_pos);

  IF a_dec > 0.0 THEN
    brake_dist := (r_vel * r_vel) / (2.0 * a_dec);
  ELSE
    brake_dist := 0.0;
  END_IF;

  IF brake_dist >= vDistance THEN
    vNewVel := r_vel - a_dec * delta_t;
    IF vNewVel < 0.0 THEN vNewVel := 0.0; END_IF;
  ELSE
    vNewVel := r_vel + a_acc * delta_t;
    IF vNewVel > r_vmax THEN vNewVel := r_vmax; END_IF;
  END_IF;

  vTravel := vNewVel * delta_t;
  IF vTravel >= vDistance THEN
    x_pos := REAL_TO_DINT(drive_target);
    v_x := 0;
    arrived := TRUE;
  ELSE
    x_pos := REAL_TO_DINT(r_pos + dir * vTravel);
    v_x := REAL_TO_DINT(vNewVel);
    arrived := FALSE;
  END_IF;
END_FUNCTION_BLOCK

(* ---- FB_SIM_ZMotion.st ---- *)
(* ============================================================
   FB_SIM_ZMotion — Vertical (Z) motion simulation

   Company : Galvatek part of the John Cockerill Group
   Author  : Jarmo Piipponen
   Created : 25.03.2026
   ============================================================
   Simulates 2D transporter lift/sink with realistic physics:
   slow start / fast middle / slow end speed profiles,
   different slow zones for wet vs dry stations.

   LIFT sequence (z_stage 2-5, 9):
     2: Slow lift    0 → ZPosSlowUp/ZPosSlowDown
     3: Fast lift    → (z_total - ZPosSlowEnd)
     4: Slow end     → z_total
     5: Dropping     at top, dripping time
     9: Drip close   drip tray close vDelay at top

   SINK sequence (z_stage 6-8):
     6: Init vDelay   (device_delay + drip_delay)
     7: Fast sink    z_total → slow_zone
     8: Slow sink    → 0 mm

   Caller sets z_stage and z_timer_s before first call.
   Output 'vDone' pulses TRUE when sequence completes.
   ------------------------------------------------------------
   Changes:
   ============================================================ *)

FUNCTION_BLOCK FB_SIM_ZMotion
VAR_INPUT
  delta_t         : REAL;    (* Cycle time in seconds — simulation internal *)
  vStationKind    : INT;     (* KIND_DRY=0, KIND_WET=1 *)
  ZPosUp          : DINT;    (* Z position at full up mm *)
  ZPosDown        : DINT;    (* Z position at full down mm *)
  ZPosSlowUp      : DINT;    (* Slow zone when going up (dry) mm *)
  ZPosSlowDown    : DINT;    (* Slow zone when going down (wet) mm *)
  ZPosSlowEnd     : DINT;    (* Slow zone at end of vTravel mm *)
  SpeedLiftSlow_Z : DINT;    (* Slow speed mm/s *)
  SpeedLiftFast_Z : DINT;    (* Fast speed mm/s *)
  DripTrayDelay   : INT;     (* Drip tray open/close vDelay ×10 = tenths of second *)
  DroppingTime    : INT;     (* Dropping/dripping time ×10 = tenths of second *)
END_VAR
VAR_IN_OUT
  z_mm      : DINT;        (* Current Z position mm *)
  z_stage   : INT;         (* Current motion stage *)
  z_timer_s : REAL;        (* Delay timer — simulation internal *)
END_VAR
VAR_OUTPUT
  vDone : BOOL;             (* TRUE when sequence complete *)
END_VAR
VAR_EXTERNAL CONSTANT
  KIND_WET : INT;
END_VAR
VAR
  (* Internal REAL copies for physics integration *)
  r_z          : REAL;
  r_total      : REAL;
  r_slow_zone  : REAL;
  r_slow_end   : REAL;
  r_slow_spd   : REAL;
  r_fast_spd   : REAL;
  r_drip       : REAL;
  r_drop       : REAL;     (* dropping/dripping time seconds *)
  z_total_mm   : DINT;     (* computed: ZPosDown - ZPosUp *)
END_VAR

  vDone := FALSE;
  z_total_mm := ZPosDown - ZPosUp;

  (* Convert DINT/INT inputs to REAL for physics *)
  r_z         := DINT_TO_REAL(z_mm);
  r_total     := DINT_TO_REAL(z_total_mm);
  r_slow_end  := DINT_TO_REAL(ZPosSlowEnd);
  r_slow_spd  := DINT_TO_REAL(SpeedLiftSlow_Z);
  r_fast_spd  := DINT_TO_REAL(SpeedLiftFast_Z);
  r_drip      := INT_TO_REAL(DripTrayDelay) / 10.0;
  r_drop      := INT_TO_REAL(DroppingTime) / 10.0;

  (* Select slow zone based on station kind *)
  IF vStationKind = KIND_WET THEN
    r_slow_zone := DINT_TO_REAL(ZPosSlowDown);
  ELSE
    r_slow_zone := DINT_TO_REAL(ZPosSlowUp);
  END_IF;

  CASE z_stage OF

    (* === LIFT: stages 2-5,9 — nosto altaasta ylös (z kasvaa: 0 → z_total) === *)
    (* Stage 1 no longer used for lift — device_delay overlaps with treatment wait *)

    2: (* Slow lift start — hidas nosto nesteestä *)
      r_z := r_z + r_slow_spd * delta_t;
      z_mm := REAL_TO_DINT(r_z);
      IF r_z >= r_slow_zone THEN
        z_stage := 3;
      END_IF;

    3: (* Fast lift — nopea nosto *)
      r_z := r_z + r_fast_spd * delta_t;
      z_mm := REAL_TO_DINT(r_z);
      IF r_z >= (r_total - r_slow_end) THEN
        z_stage := 4;
      END_IF;

    4: (* Slow lift end — hidas loppunosto *)
      r_z := r_z + r_slow_spd * delta_t;
      IF r_z >= r_total THEN
        z_mm := z_total_mm;
        z_timer_s := r_drop;
        z_stage := 5;
      ELSE
        z_mm := REAL_TO_DINT(r_z);
      END_IF;

    5: (* Dropping / dripping — valutusaika yläasemassa *)
      z_timer_s := z_timer_s - delta_t;
      IF z_timer_s <= 0.0 THEN
        z_timer_s := r_drip;
        z_stage := 9;
      END_IF;

    9: (* Drip tray close — tippakouru sulkeutuu *)
      z_timer_s := z_timer_s - delta_t;
      IF z_timer_s <= 0.0 THEN
        z_stage := 0;
        vDone := TRUE;
      END_IF;

    (* === SINK: stages 6-8 — lasku altaaseen (z pienenee: z_total → 0) === *)

    6: (* Init vDelay: device_delay + drip_delay *)
      z_timer_s := z_timer_s - delta_t;
      IF z_timer_s <= 0.0 THEN
        z_stage := 7;
      END_IF;

    7: (* Fast sink — nopea lasku *)
      r_z := r_z - r_fast_spd * delta_t;
      z_mm := REAL_TO_DINT(r_z);
      IF r_z <= r_slow_zone THEN
        z_stage := 8;
      END_IF;

    8: (* Slow sink — hidas lasku nesteeseen *)
      r_z := r_z - r_slow_spd * delta_t;
      IF r_z <= 0.0 THEN
        z_mm := 0;
        z_stage := 0;
        vDone := TRUE;
      ELSE
        z_mm := REAL_TO_DINT(r_z);
      END_IF;

  END_CASE;

END_FUNCTION_BLOCK

(* ---- SIM_FB_ClearConfig.st ---- *)
(* ============================================================
   SIM_FB_ClearConfig — Clear all PLC configuration data

   Company : Galvatek part of the John Cockerill Group
   Author  : Jarmo Piipponen
   Created : 25.03.2026
   ============================================================
   Called by PLC_PRG when Gateway sends cmd=3 (clear_all).
   Zeroes out all stations, transporter configs, transporter
   states and units so the PLC is ready for fresh config upload.
   ------------------------------------------------------------
   Changes:
   ============================================================ *)

FUNCTION_BLOCK SIM_FB_ClearConfig
VAR_EXTERNAL CONSTANT
    MAX_Transporters    : INT;
    MAX_STATIONS_PER_STEP       : INT;
    MAX_STEPS_PER_PROGRAM       : INT;
    MAX_TASK_QUEUE      : INT;
    MIN_StationIndex : INT;
    MAX_StationIndex   : INT;
    MAX_Units           : INT;
    DEP_MAX_WAITING     : INT;
    NOT_PROCESSED       : INT;
END_VAR

VAR_EXTERNAL
  CountStations       : INT;
  Stations         : ARRAY[MIN_StationIndex..MAX_StationIndex] OF UDT_StationType;
  g_station_occupancy     : ARRAY[1..MAX_StationIndex] OF UDT_JC_UnitAtStationType;
  Transporters              : ARRAY[0..MAX_Transporters] OF UDT_TransporterType;
  g_transporter      : ARRAY[1..MAX_Transporters] OF UDT_TransporterStatusType;
  g_sim_trans        : ARRAY[1..MAX_Transporters] OF UDT_JC_SimTransporterType;
  g_dispatched_task  : ARRAY[1..MAX_Transporters] OF UDT_JC_DispatchedTaskType;
  g_unit            : ARRAY[1..MAX_Units] OF UDT_JC_UnitType;
  g_ntt             : ARRAY[1..MAX_Transporters] OF UDT_JC_NttTransporterType;
  g_batch          : ARRAY[1..MAX_Units] OF UDT_BatchType;
  TreatmentPrograms         : ARRAY[1..MAX_Units] OF UDT_TreatmentProgramType;
  g_avoid_status     : ARRAY[MIN_StationIndex..MAX_StationIndex] OF INT;
  g_schedule         : ARRAY[1..MAX_Units] OF UDT_JC_TskScheduleType;
  g_task             : ARRAY[1..MAX_Transporters] OF UDT_JC_TskQueueType;
  g_sim_ui_schedule  : ARRAY[1..MAX_Units] OF UDT_JC_TskScheduleType;
  g_sim_ui_task      : ARRAY[1..MAX_Transporters] OF UDT_JC_TskQueueType;
  g_sim_ui_wait_unit : INT;
  g_sim_ui_wait_reason : INT;
  g_dep_pending      : UDT_JC_DepPendingWriteType;
  g_dep_activated    : BOOL;
  g_tsk_stable       : BOOL;
  g_dep_waiting_count : INT;
  g_dep_waiting       : ARRAY[1..DEP_MAX_WAITING] OF INT;
END_VAR
VAR
  i : INT;
  j : INT;
  k : INT;
END_VAR

(* --- Clear all stations --- *)
FOR i := MIN_StationIndex TO MAX_StationIndex DO
  Stations[i].TankId       := 0;
  Stations[i].IsInUse       := FALSE;
  Stations[i].XPosition    := 0;
  Stations[i].YPosition    := 0;
  Stations[i].ZPosition    := 0;
  Stations[i].DryWet          := 0;
  Stations[i].StationType     := 0;
  Stations[i].DrippingTime := 0;
  Stations[i].DeviceDelay  := 0;
END_FOR;

(* --- Clear all location tracking (transporters 1..MAX_Transporters + stations MIN..MAX) --- *)
FOR i := 1 TO MAX_StationIndex DO
  g_station_occupancy[i].UnitId     := 0;
  g_station_occupancy[i].ChangeTime := 0;
END_FOR;
CountStations := 0;

(* --- Clear all transporter configs --- *)
FOR i := 1 TO MAX_Transporters DO
  Transporters[i].DrivePosMin   := 0;
  Transporters[i].DrivePosMax   := 0;
  Transporters[i].YMinDriveLimit   := 0;
  Transporters[i].YMaxDriveLimit   := 0;
  Transporters[i].CollisionWidth    := 0;
  Transporters[i].AvoidanceWidth    := 0;
  Transporters[i].Acceleration_X     := 0;
  Transporters[i].Deceleration_X     := 0;
  Transporters[i].SpeedMax_X    := 0;
  Transporters[i].ZPosDown    := 0;
  Transporters[i].ZPosSlowUp := 0;
  Transporters[i].ZPosSlowDown := 0;
  Transporters[i].ZPosSlowEnd := 0;
  Transporters[i].SpeedLiftSlow_Z   := 0;
  Transporters[i].SpeedLiftFast_Z   := 0;
  Transporters[i].DripTrayDelay  := 0;
  FOR j := 1 TO 4 DO
    Transporters[i].TaskArea[j].MinLift := 0;
    Transporters[i].TaskArea[j].MaxLift := 0;
    Transporters[i].TaskArea[j].MinSink := 0;
    Transporters[i].TaskArea[j].MaxSink := 0;
  END_FOR;
END_FOR;

(* --- Clear avoid status --- *)
FOR i := MIN_StationIndex TO MAX_StationIndex DO
  g_avoid_status[i] := 0;
END_FOR;

(* --- Clear all transporter states --- *)
FOR i := 1 TO MAX_Transporters DO
  g_transporter[i].IsActive          := FALSE;
  g_transporter[i].Status          := 0;
  g_transporter[i].Phase           := 0;
  g_transporter[i].TaskId         := 0;
  g_transporter[i].LiftStationTarget    := 0;
  g_transporter[i].SinkStationTarget    := 0;
  g_transporter[i].DrippingTime   := 0;
  g_transporter[i].TaskRemainingTime  := 0;
  g_transporter[i].CurrentStation := 0;
  g_transporter[i].XFinalTarget  := 0;
  g_transporter[i].XDriveTarget  := 0;
  g_transporter[i].YFinalTarget  := 0;
  g_transporter[i].YDriveTarget  := 0;
  g_transporter[i].XPosition            := 0;
  g_transporter[i].YPosition            := 0;
  g_transporter[i].ZPosition            := 0;
  g_sim_trans[i].XVelocity           := 0;
  g_sim_trans[i].ZStage         := 0;
  g_sim_trans[i].ZTimer       := 0.0;
  g_transporter[i].IdleStartTime := g_time_s;  (* prevent spurious move-away after clear *)
  g_dispatched_task[i].Active := FALSE;
  g_transporter[i].XMinDriveLimit     := 0;
  g_transporter[i].XMaxDriveLimit     := 0;
END_FOR;

(* --- Clear all units --- *)
FOR i := 1 TO MAX_Units DO
  g_unit[i].location := 0;
  g_unit[i].Status   := 0;
  g_unit[i].Target   := 0;
END_FOR;

(* --- Clear NTT destinations --- *)
FOR i := 1 TO MAX_Transporters DO
  FOR j := 1 TO 8 DO
    g_ntt[i].Target[j].StationCount := 0;
    g_ntt[i].Target[j].FallbackCount := 0;
    FOR k := 1 TO MAX_STATIONS_PER_STEP DO
      g_ntt[i].Target[j].Stations[k] := 0;
      g_ntt[i].Target[j].FallbackStations[k] := 0;
    END_FOR;
  END_FOR;
END_FOR;

(* --- Clear all batches --- *)
FOR i := 1 TO MAX_Units DO
  g_batch[i].BatchCode  := 0;
  g_batch[i].State       := 0;
  g_batch[i].ProgId     := 0;
  g_batch[i].CurStage   := 0;
  g_batch[i].MinTime    := 0;
  g_batch[i].MaxTime    := 0;
  g_batch[i].CalTime    := 0;
  g_batch[i].StartTime  := LINT#0;
END_FOR;

(* --- Clear all treatment programs --- *)
FOR i := 1 TO MAX_Units DO
  TreatmentPrograms[i].ProgramId := 0;
  TreatmentPrograms[i].ProgramName := '';
  TreatmentPrograms[i].StepCount := 0;
  FOR j := 0 TO MAX_STEPS_PER_PROGRAM DO
    FOR k := 0 TO 4 DO
      TreatmentPrograms[i].Steps[j].Stations[k] := 0;
    END_FOR;
    TreatmentPrograms[i].Steps[j].StationCount := 0;
    TreatmentPrograms[i].Steps[j].MinTime := 0;
    TreatmentPrograms[i].Steps[j].MaxTime := 0;
    TreatmentPrograms[i].Steps[j].CalTime := 0;
  END_FOR;
END_FOR;

(* --- Clear all schedules (g_schedule) --- *)
FOR i := 1 TO MAX_Units DO
  g_schedule[i].StageCount := 0;
  FOR j := 0 TO MAX_STEPS_PER_PROGRAM DO
    g_schedule[i].Stages[j].station       := 0;
    g_schedule[i].Stages[j].EntryTime    := 0;
    g_schedule[i].Stages[j].ExitTime     := 0;
    g_schedule[i].Stages[j].MinTime      := 0;
    g_schedule[i].Stages[j].CalcTime     := 0;
    g_schedule[i].Stages[j].MaxTime      := 0;
    g_schedule[i].Stages[j].TransferTime := 0;
  END_FOR;
END_FOR;

(* --- Clear all task queues (g_task) --- *)
FOR i := 1 TO MAX_Transporters DO
  g_task[i].Count := 0;
  FOR j := 1 TO MAX_TASK_QUEUE DO
    g_task[i].Queue[j].Unit         := 0;
    g_task[i].Queue[j].Stage        := 0;
    g_task[i].Queue[j].LiftStationTarget := 0;
    g_task[i].Queue[j].SinkStationTarget := 0;
    g_task[i].Queue[j].StartTime   := 0;
    g_task[i].Queue[j].FinishTime  := 0;
    g_task[i].Queue[j].CalcTime    := 0;
    g_task[i].Queue[j].MinTime     := 0;
    g_task[i].Queue[j].MaxTime     := 0;
  END_FOR;
END_FOR;

(* --- Clear UI snapshot --- *)
FOR i := 1 TO MAX_Units DO
  g_sim_ui_schedule[i].StageCount := 0;
END_FOR;
FOR i := 1 TO MAX_Transporters DO
  g_sim_ui_task[i].Count := 0;
END_FOR;
g_sim_ui_wait_unit := 0;
g_sim_ui_wait_reason := 0;

(* --- Clear departure pending write --- *)
g_dep_pending.Valid := FALSE;
g_dep_pending.BatchUnit  := 0;
g_dep_pending.BatchStage := 0;
g_dep_pending.BatchState := NOT_PROCESSED;

(* --- Clear departure scheduler state (previously missing) --- *)
g_dep_activated     := FALSE;
g_tsk_stable        := TRUE;   (* JS: tasksStableFlag starts true on empty line *)
g_dep_waiting_count := 0;
FOR i := 1 TO 5 DO
  g_dep_waiting[i] := 0;
END_FOR;

END_FUNCTION_BLOCK

(* ---- SIM_FB_EventQueue.st ---- *)
(* ============================================================
   SIM_FB_EventQueue — Event message queue handler (OPC UA)

   Company : Galvatek part of the John Cockerill Group
   Author  : Jarmo Piipponen
   Created : 25.03.2026
   ============================================================
   Manages a circular 10-slot event queue (Event).

   Enqueue: caller writes msg to EventPending, sets
   EventPendingValid := TRUE. This FB picks it up.

   Dequeue: Gateway reads Event.Buffer[Head] via OPC UA,
   then writes EventAckSeq to acknowledge.

   Called every PLC scan from PLC_PRG.
   ------------------------------------------------------------
   Changes:
   ============================================================ *)

FUNCTION_BLOCK SIM_FB_EventQueue
VAR_EXTERNAL
  Event               : UDT_JC_EventQueueType;
  EventPending       : UDT_JC_EventMsgType;
  EventPendingValid : BOOL;
  EventAckSeq       : INT;
END_VAR
VAR
  vTail : INT;
END_VAR

(* ── 1. Enqueue: pick up pending message if queue not full ── *)
IF EventPendingValid AND Event.Count < 10 THEN
  vTail := ((Event.Head - 1 + Event.Count) MOD 10) + 1;

  EventPending.Seq := Event.NextSeq;
  Event.NextSeq := Event.NextSeq + 1;
  IF Event.NextSeq > 32000 THEN
    Event.NextSeq := 1;
  END_IF;

  Event.Buffer[vTail] := EventPending;
  Event.Count := Event.Count + 1;

  EventPendingValid := FALSE;
END_IF;

(* ── 2. Dequeue: check gateway ack for head message ── *)
IF Event.Count > 0 THEN
  IF EventAckSeq = Event.Buffer[Event.Head].Seq THEN
    Event.Head := (Event.Head MOD 10) + 1;
    Event.Count := Event.Count - 1;
  END_IF;
END_IF;

END_FUNCTION_BLOCK

(* ---- SIM_FB_MainCycle.st ---- *)
(* ===========================================================================================
 *  SIM_FB_MainCycle — Simulator main cycle (all SIM-specific logic)
 *
 *  Company : Galvatek part of the John Cockerill Group
 *  Author  : Jarmo Piipponen
 *  Created : 08.04.2026
 *
 * -------------------------------------------------------------------------------------------
 *  Encapsulates everything that is simulation-only and NOT needed in production:
 *    - OPC UA command handler (init / clear)
 *    - System time calculation (g_time_s via offset from gateway sync)
 *    - TWA calculation
 *    - Physics simulation (delta_t + SIM_FB_RunTasks)
 *    - UI schedule snapshot for gateway
 *    - Event queue processing
 *
 *  In production PLC_PRG, this FB is removed entirely.
 *  PLC_PRG only needs: time from real PLC clock, TWA, MainScheduler.
 * ========================================================================================= *)

FUNCTION_BLOCK SIM_FB_MainCycle

(* Introduction of Variables ----------------------------------------------------------------*)

VAR_EXTERNAL CONSTANT
    MAX_TRANSPORTERS        : INT;
    MAX_STATIONS_PER_STEP   : INT;
    MIN_STATION_INDEX        : INT;
    MAX_STATION_INDEX        : INT;
    MAX_UNITS               : INT;
    DEP_MAX_WAITING         : INT;
END_VAR

VAR_EXTERNAL
  CountStations             : INT;
  Stations                  : ARRAY[MIN_STATION_INDEX..MAX_STATION_INDEX] OF UDT_StationType;
  g_station_occupancy       : ARRAY[1..MAX_STATION_INDEX] OF UDT_JC_UnitAtStationType;
  Transporters              : ARRAY[0..MAX_TRANSPORTERS] OF UDT_TransporterType;
  g_transporter             : ARRAY[1..MAX_TRANSPORTERS] OF UDT_TransporterStatusType;
  g_sim_trans               : ARRAY[1..MAX_TRANSPORTERS] OF UDT_JC_SimTransporterType;
  g_unit                    : ARRAY[1..MAX_UNITS] OF UDT_JC_UnitType;
  g_ntt                     : ARRAY[1..MAX_TRANSPORTERS] OF UDT_JC_NttTransporterType;
  g_batch                   : ARRAY[1..MAX_UNITS] OF UDT_BatchType;
  TreatmentPrograms         : ARRAY[1..MAX_UNITS] OF UDT_TreatmentProgramType;
  g_avoid_status            : ARRAY[MIN_STATION_INDEX..MAX_STATION_INDEX] OF INT;
  g_move                    : ARRAY[1..MAX_TRANSPORTERS] OF UDT_JC_MoveTimesType;
  g_schedule                : ARRAY[1..MAX_UNITS] OF UDT_JC_TskScheduleType;
  g_task                    : ARRAY[1..MAX_TRANSPORTERS] OF UDT_JC_TskQueueType;
  g_dep_activated           : BOOL;
  g_tsk_stable              : BOOL;
  g_dep_waiting_count       : INT;
  g_dep_overlap             : UDT_JC_DepOverlapType;
  g_dep_pending             : UDT_JC_DepPendingWriteType;
  g_dep_waiting             : ARRAY[1..DEP_MAX_WAITING] OF INT;
  g_sched_dbg_tsk_phase     : INT;
  g_sched_dbg_dep_phase     : INT;
  g_sim_ui_schedule         : ARRAY[1..MAX_UNITS] OF UDT_JC_TskScheduleType;
  g_sim_ui_task             : ARRAY[1..MAX_TRANSPORTERS] OF UDT_JC_TskQueueType;
  g_sim_ui_wait_unit        : INT;
  g_sim_ui_wait_reason      : INT;
  g_sched_dbg_turn          : INT;
  g_conflict_resolved       : BOOL;
  g_sched_dbg_batch_cnt     : INT;
  g_time_s                  : LINT;
  g_time_100ms              : LINT;
  g_time_offset             : LINT;
  g_time_sync               : LINT;
  g_event                   : UDT_JC_EventQueueType;
  g_event_pending           : UDT_JC_EventMsgType;
  g_event_pending_valid     : BOOL;
  g_event_ack_seq           : INT;
  g_cmd_code                : INT;
  g_cmd_param               : INT;
  g_sched_dbg_dep_cur_wait_unit : INT;
END_VAR

VAR_OUTPUT
  o_init_done               : BOOL;
END_VAR

VAR
  init_done                 : BOOL := FALSE;
  i                         : INT;
  clear_cfg                 : SIM_FB_ClearConfig;
  run_tasks                 : SIM_FB_RunTasks;
  evt_queue                 : SIM_FB_EventQueue;
  now_ms                    : LINT := 0;
  prev_ms                   : UDINT := 0;
  sim_delta_t               : REAL := 0.02;
  prev_tsk_phase            : INT := 0;
  prev_dep_phase            : INT := 0;
END_VAR

(* ============================================================
   COMMAND HANDLER — OPC UA (direct, no sequence handshake)
   Gateway writes g_cmd_code + g_cmd_param in one atomic OPC UA
   call. PLC processes when g_cmd_code <> 0 and clears it.
   ============================================================ *)
IF g_cmd_code <> 0 THEN

  IF g_cmd_code = 3 THEN
    (* ── Clear all config data ── *)
    clear_cfg();
    init_done := FALSE;
    CountStations := 0;

  ELSIF g_cmd_code = 2 THEN
    (* ── Finish init: all config already uploaded via OPC UA ── *)
    CountStations := g_cmd_param;

    FOR i := 1 TO MAX_TRANSPORTERS DO
      IF Transporters[i].TaskArea[1].MinLift > 0 THEN
        g_transporter[i].IsActive := TRUE;
        g_transporter[i].Status := 3;  (* auto_idle *)
      ELSE
        g_transporter[i].IsActive := FALSE;
        g_transporter[i].Status := 0;  (* not_used *)
      END_IF;
      g_transporter[i].Phase := 0;
      g_sim_trans[i].ZStage := 0;
      g_sim_trans[i].XVelocity := 0;
      g_sim_trans[i].ZTimer := 0.0;
      g_transporter[i].IdleStartTime := g_time_s;
      g_transporter[i].XMinDriveLimit := Transporters[i].DrivePosMin;
      g_transporter[i].XMaxDriveLimit := Transporters[i].DrivePosMax;

      (* Start position: at own area minimum, z=0 *)
      g_transporter[i].XPosition := Transporters[i].DrivePosMin;
      g_transporter[i].ZPosition := 0;
      g_transporter[i].CurrentStation := 0;
    END_FOR;

    init_done := TRUE;

    (* Calculate time offset: real unix time - uptime *)
    g_time_offset := g_time_sync - UDINT_TO_LINT(SysTimeGetMs()) / 1000;

    (* Build g_station_occupancy from g_unit[].location so SIM_FB_RunTasks
       can find units on stations via g_station_occupancy[stn].UnitId.
       Gateway writes g_unit[] but not g_station_occupancy[]. *)
    FOR i := 1 TO MAX_UNITS DO
      IF g_unit[i].location >= MIN_STATION_INDEX
         AND g_unit[i].location <= MAX_STATION_INDEX THEN
        g_station_occupancy[g_unit[i].location].UnitId     := i;
        g_station_occupancy[g_unit[i].location].ChangeTime  := g_time_s;
      END_IF;
    END_FOR;

    (* Init event queue *)
    g_event.Head := 1;
    g_event.NextSeq := 1;
    g_event.Count := 0;
  END_IF;

  g_cmd_code := 0;  (* Command processed — clear trigger *)
END_IF;

(* ============================================================
   MAIN TRANSPORT CYCLE — only runs when init_done
   ============================================================ *)
IF init_done THEN

  (* ── System time: uptime + offset = real unix seconds ── *)
  now_ms := UDINT_TO_LINT(SysTimeGetMs());
  g_time_s := g_time_offset + now_ms / 1000;        (* seconds, unix epoch *)
  g_time_100ms := g_time_offset * 10 + now_ms / 100; (* 0.1s ticks, unix epoch *)

  (* ── Actual cycle time for physics simulation ── *)
  IF prev_ms > 0 THEN
    sim_delta_t := UDINT_TO_REAL(LINT_TO_UDINT(now_ms) - prev_ms) / 1000.0;
  END_IF;
  prev_ms := LINT_TO_UDINT(now_ms);

  (* ── Execute transporter tasks (physics simulation) ── *)
  run_tasks(i_run := init_done, i_delta_t := sim_delta_t);

END_IF;  (* init_done *)

o_init_done := init_done;

(* ── UI schedule snapshot — copy stable data for gateway reads ── *)
IF g_sched_dbg_tsk_phase = 10000 AND prev_tsk_phase <> 10000 THEN
  g_sim_ui_schedule := g_schedule;
  g_sim_ui_task     := g_task;
END_IF;
IF g_sched_dbg_dep_phase = 8000 AND prev_dep_phase <> 8000 THEN
  g_sim_ui_wait_unit   := 0;
  g_sim_ui_wait_reason := 0;
END_IF;
IF g_sched_dbg_dep_phase = 9000 AND prev_dep_phase <> 9000 THEN
  g_sim_ui_wait_unit   := g_sched_dbg_dep_cur_wait_unit;
  g_sim_ui_wait_reason := 1;
END_IF;
prev_tsk_phase := g_sched_dbg_tsk_phase;
prev_dep_phase := g_sched_dbg_dep_phase;

(* ── Event queue — always runs, not gated by init_done ── *)
evt_queue();

END_FUNCTION_BLOCK
